{attribute 'linkalways'} 
{attribute 'no_explicit_call' := 'This FB is a CLASS and must be accessed using methods or properties'}
{attribute 'enable_dynamic_creation'}
FUNCTION_BLOCK Content EXTENDS Disposable IMPLEMENTS I_Content
VAR
	_name : T_MAXSTRING;
	_data : I_Datatype;
	_parent : I_HaveContent;
END_VAR

METHOD PUBLIC Accept
VAR_INPUT
	Visitor : I_ContentVisitor;
END_VAR
Visitor.VisitContent(this^);
END_METHOD

PROPERTY PUBLIC Data : I_DataType
GET
Data := _data;
END_GET
END_PROPERTY

METHOD FB_init : BOOL
VAR_INPUT
	bInitRetains : BOOL; // if TRUE, the retain variables are initialized (warm start / cold start)
	bInCopyCode : BOOL;  // if TRUE, the instance afterwards gets moved into the copy code (online change)
	Name : T_MAXSTRING;
	Data : I_Datatype;
	Parent : I_HaveContent;
END_VAR
_name := Name;
_data := Data;
RegisterWithParent(Parent);
END_METHOD

PROPERTY PUBLIC Name : T_MAXSTRING
GET
Name := _name;
END_GET
END_PROPERTY

PROPERTY PUBLIC Parent : I_HaveContent
GET
Parent := _parent;
END_GET
END_PROPERTY

METHOD PUBLIC RegisterWithParent
VAR_INPUT
	Parent : I_HaveContent;
END_VAR
IF Parent = 0 THEN
	RETURN;
END_IF

THIS^._parent := Parent;
Parent.AddContent(THIS^);
END_METHOD

METHOD PUBLIC SerializeWith
VAR_INPUT
	Serializer : I_Serializer;
END_VAR
// make a content object.
// content name
// make a key called value, put _data in that

_data.SerializeWith(Serializer);
END_METHOD

END_FUNCTION_BLOCK

(* stored: Version 1.1.0.1, ProductVersion 3.1.4024.12
   POU Content: Id {0d9cf418-5c17-01af-15e9-b437781a1d71}, SpecialFunc None
   Folder Constructor: Id {837d23f4-e080-04af-1c00-afd1f5791c19}
   Method Accept: Id {4deecd26-05a3-087a-0d9b-39d9f2ed6081}
   Property Data: Id {84f51fb0-45ab-000a-2b80-8ac17966921c}
   Get Get: Id {4a624fc3-292a-0b2c-3065-c19a38ab6b07}
   Method FB_init: Id {2d9dcb5d-b2bf-00b6-3905-b549a314f45c}
   Property Name: Id {e0fe422f-2992-0a7a-3a67-4d74882b6ea4}
   Get Get: Id {6e49c007-b4a0-041b-1088-5b57730553f3}
   Property Parent: Id {2024bed4-f17f-0a30-1b47-bca1f219aa82}
   Get Get: Id {5956cbec-13e7-03c8-3e5e-1d37acadef69}
   Method RegisterWithParent: Id {5e8e70e3-cedb-09b8-1c96-4b1b0a7fd098}
   Method SerializeWith: Id {d6dbce2b-9fc3-4a10-9518-677d2589af3a} *)
